// TwinCAT 3 PLC project PLC1
// ProgramVersion: 3.1.4020.4
// libraries:
//   Tc2_Standard, * (Beckhoff Automation GmbH)
//   Tc2_System, * (Beckhoff Automation GmbH)
//   Tc3_Module, * (Beckhoff Automation GmbH)
// project tree:
//   GVLs/ Grinder.TcGVL
//   / PlcTask.TcTTO
//   POUs/ MAIN.TcPOU, RunGrindingWheel.TcPOU
// real-time tasks:
//   TASK PlcTask: cycle T#10ms, priority 20, ADS port 350
// I/O:
//   DEVICE Device 1 (EtherCAT), AmsNetId 10.175.62.142.2.1
//     Box 3 (XMC_ESC) [XMC_ESC]
//     Box 4 (XMC_ESC) [XMC_ESC]
// variable links:
//   PLC1/PLC1 Instance <-> Device 1 (EtherCAT)/Box 3 (XMC_ESC)
//     PlcTask Inputs/Grinder.StartGrindingWheelPB <-> IN_GENERIC process data mapping/IN_GEN_Bit1
//     PlcTask Inputs/Grinder.StopGrindingWheelPB <-> IN_GENERIC process data mapping/IN_GEN_Bit2
//   PLC1/PLC1 Instance <-> Device 1 (EtherCAT)/Box 4 (XMC_ESC)
//     PlcTask Outputs/Grinder.GrindingsWheelMS <-> OUT_GENERIC process data mapping/OUT_GEN_Bit1

CONFIGURATION PLC1
    RESOURCE PLC ON TwinCAT3
        TASK PlcTask(INTERVAL := T#10ms, PRIORITY := 20);
        PROGRAM MAIN WITH PlcTask : MAIN;
    END_RESOURCE
END_CONFIGURATION

// ---- GVLs/Grinder.TcGVL
{attribute 'qualified_only'}
VAR_GLOBAL
  GrindingsWheelMS       AT %Q* : BOOL;
  StartGrindingWheelPB   AT %I* : BOOL;
  StopGrindingWheelPB    AT %I* : BOOL;

END_VAR

// ---- POUs/MAIN.TcPOU
PROGRAM MAIN
VAR
END_VAR

RunGrindingWheel();

END_PROGRAM

// ---- POUs/RunGrindingWheel.TcPOU
PROGRAM RunGrindingWheel
VAR
END_VAR

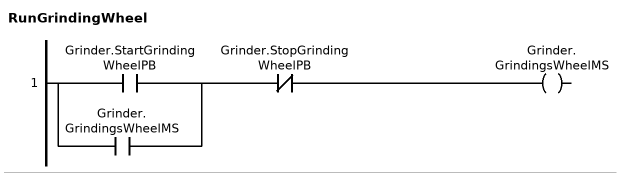
// NETWORK 1
Grinder.GrindingsWheelMS := (Grinder.StartGrindingWheelPB OR Grinder.GrindingsWheelMS) AND NOT Grinder.StopGrindingWheelPB;

END_PROGRAM
